(* IEC 61131-3 sources: AXOpen/src/components.newlibrary/app/src/Documentation, 1 file *)

(* ---- DocumentationContext.st ---- *)
CLASS DocumentationContext EXTENDS AXOpen.Core.AxoContext
    VAR PUBLIC
        cylinder : Component;
    END_VAR

    METHOD PROTECTED OVERRIDE Main
        cylinder.Run(THIS);
    END_METHOD
END_CLASS
